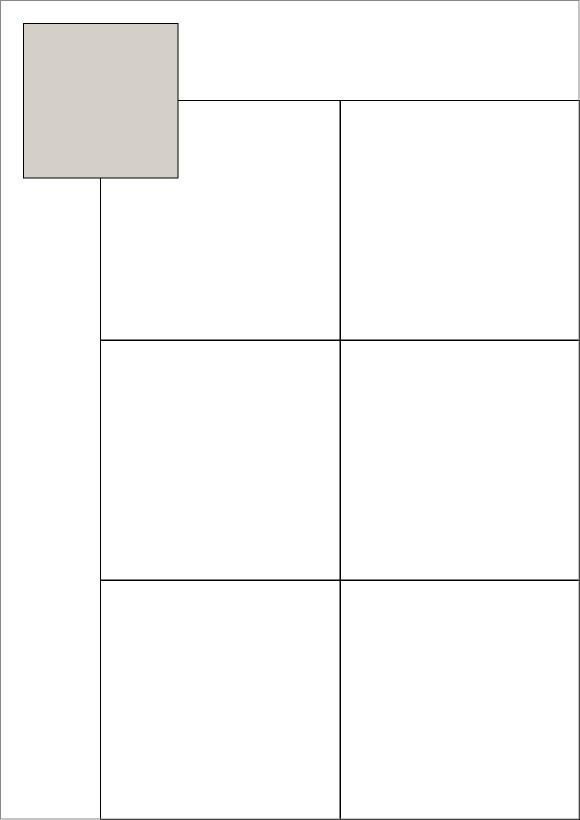
VISUALIZATION Visualization  // 580x820
    Rectangle (100,100 240x240)
    Rectangle (340,100 240x240)
    Rectangle (100,340 240x240)
    Rectangle (340,340 240x240)
    Rectangle (100,580 240x240)
    Rectangle (340,580 240x240)
    RoundedRectangle (23,23 155x155)
END_VISUALIZATION

(* stored: Version 1.1.0.1, ProductVersion 3.1.4024.12
   Visu Visualization: Id {8b240b3a-e04f-48cf-9364-903e534853d6} *)
